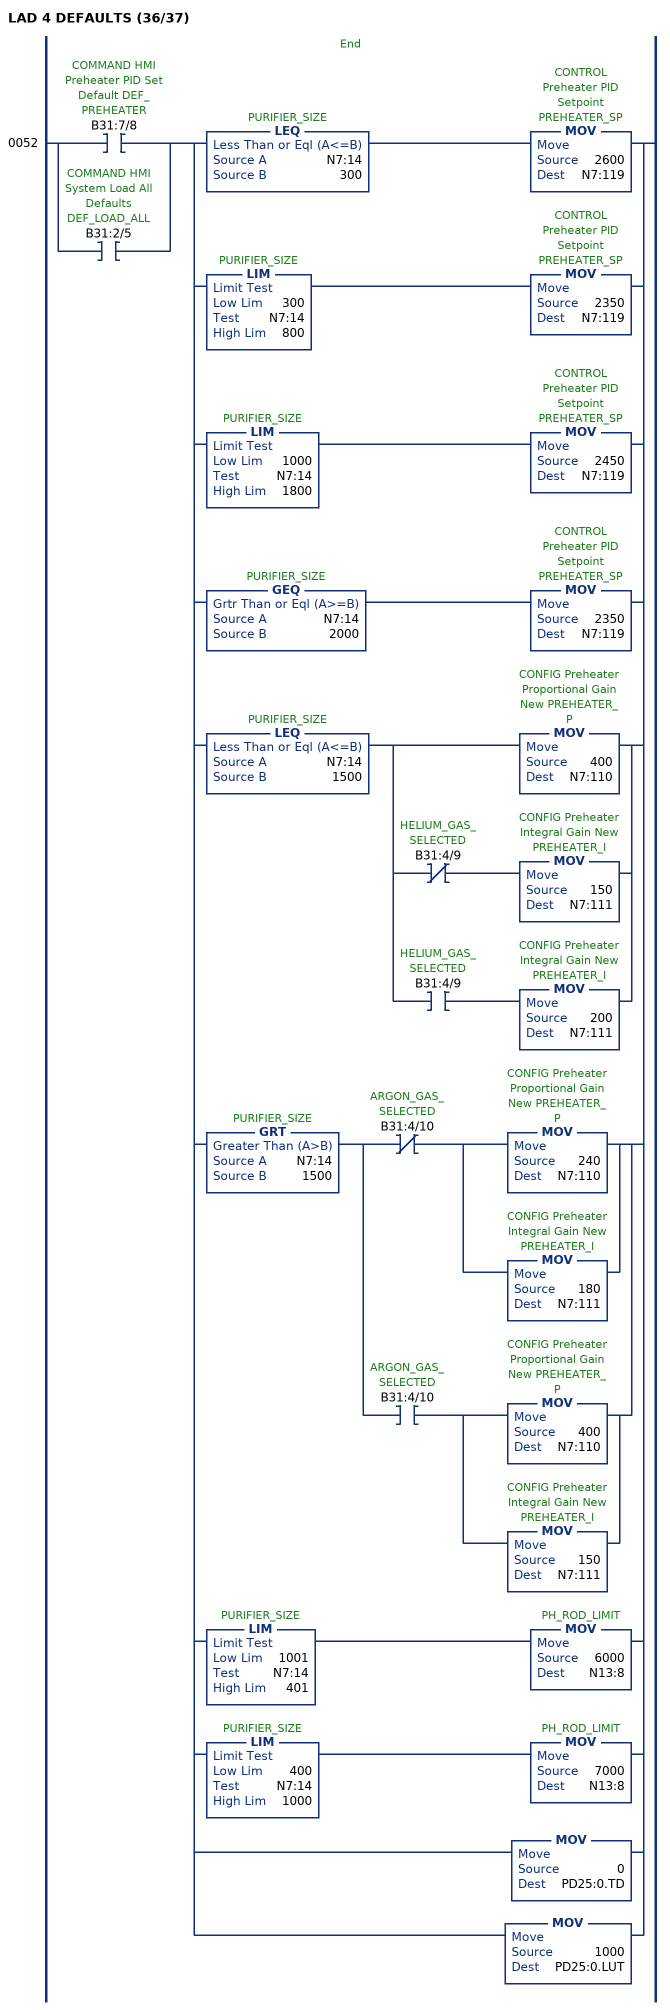
% Rung: 52 %
% End %
SOR BST XIC B31:7/8 NXB XIC B31:2/5 BND BST BST LEQ N7:14 300 MOV 2600 N7:119 NXB LIM 300 N7:14 800 MOV 2350 N7:119 NXB LIM 1000 N7:14 1800 MOV 2450 N7:119 NXB GEQ N7:14 2000 MOV 2350 N7:119 BND NXB BST LEQ N7:14 1500 BST MOV 400 N7:110 NXB BST XIO B31:4/9 MOV 150 N7:111 NXB XIC B31:4/9 MOV 200 N7:111 BND BND NXB GRT N7:14 1500 BST XIO B31:4/10 BST MOV 240 N7:110 NXB MOV 180 N7:111 BND NXB XIC B31:4/10 BST MOV 400 N7:110 NXB MOV 150 N7:111 BND BND BND NXB BST LIM 1001 N7:14 401 MOV 6000 N13:8 NXB LIM 400 N7:14 1000 MOV 7000 N13:8 BND NXB MOV 0 PD25:0.TD NXB MOV 1000 PD25:0.LUT BND EOR
%   B31:7/8  DEF_PREHEATER  "COMMAND HMI Preheater PID Set Default" %
%   B31:2/5  DEF_LOAD_ALL  "COMMAND HMI System Load All Defaults" %
%   N7:14  PURIFIER_SIZE %
%   N7:119  PREHEATER_SP  "CONTROL Preheater PID Setpoint" %
%   N7:110  PREHEATER_P  "CONFIG Preheater Proportional Gain New" %
%   B31:4/9  HELIUM_GAS_SELECTED %
%   N7:111  PREHEATER_I  "CONFIG Preheater Integral Gain New" %
%   B31:4/10  ARGON_GAS_SELECTED %
%   N13:8  PH_ROD_LIMIT %

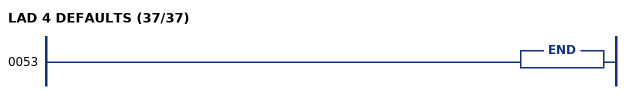
% Rung: 53 %
SOR END EOR

LADDER 5 "SYS_FAULTS"    % Monitors the system fault conditions %
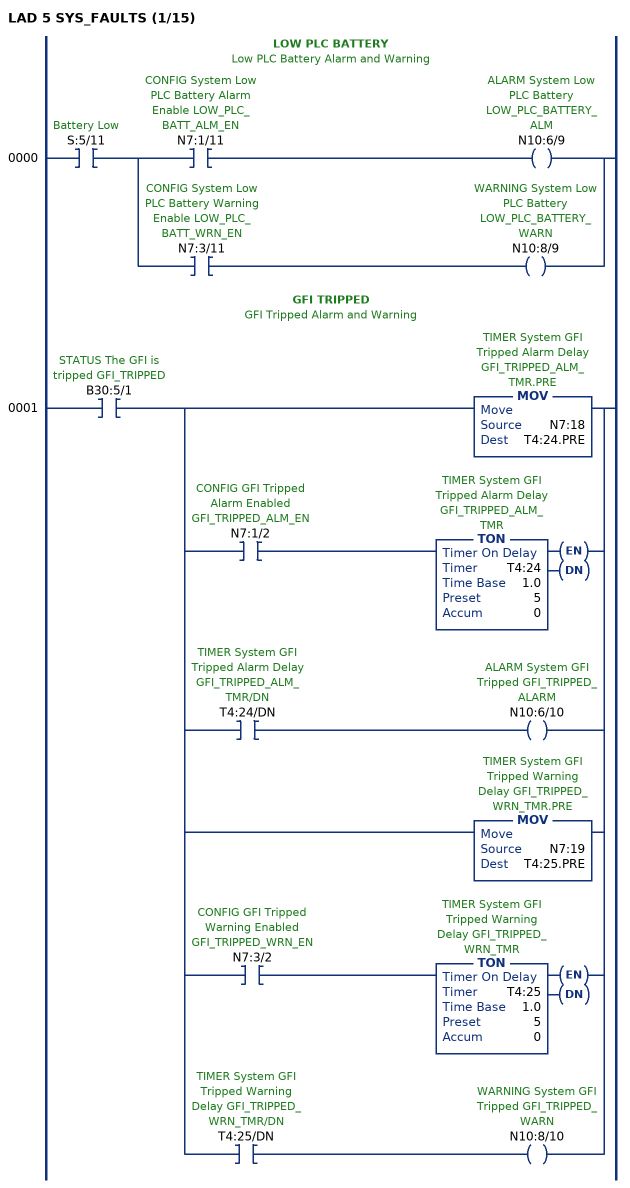
% Rung: 0 %
% TITLE: LOW PLC BATTERY %
% Low PLC Battery Alarm and Warning %
SOR XIC S:5/11 BST XIC N7:1/11 OTE N10:6/9 NXB XIC N7:3/11 OTE N10:8/9 BND EOR
%   S:5/11  "Battery Low" %
%   N7:1/11  LOW_PLC_BATT_ALM_EN  "CONFIG System Low PLC Battery Alarm Enable" %
%   N10:6/9  LOW_PLC_BATTERY_ALM  "ALARM System Low PLC Battery" %
%   N7:3/11  LOW_PLC_BATT_WRN_EN  "CONFIG System Low PLC Battery Warning Enable" %
%   N10:8/9  LOW_PLC_BATTERY_WARN  "WARNING System Low PLC Battery" %
% Rung: 1 %
% TITLE: GFI TRIPPED %
% GFI Tripped Alarm and Warning %
SOR XIC B30:5/1 BST MOV N7:18 T4:24.PRE NXB XIC N7:1/2 TON T4:24 1.0 5 0 NXB XIC T4:24/DN OTE N10:6/10 NXB MOV N7:19 T4:25.PRE NXB XIC N7:3/2 TON T4:25 1.0 5 0 NXB XIC T4:25/DN OTE N10:8/10 BND EOR
%   B30:5/1  GFI_TRIPPED  "STATUS The GFI is tripped" %
%   N7:18  GFI_TRIPPED_ALM_DLY  "CONFIG GFI fault alarm delay" %
%   T4:24  GFI_TRIPPED_ALM_TMR  "TIMER System GFI Tripped Alarm Delay" %
%   N7:1/2  GFI_TRIPPED_ALM_EN  "CONFIG GFI Tripped Alarm Enabled" %
%   N10:6/10  GFI_TRIPPED_ALARM  "ALARM System GFI Tripped" %
%   N7:19  GFI_TRIPPED_WRN_DLY  "CONFIG GFI fault warning delay" %
%   T4:25  GFI_TRIPPED_WRN_TMR  "TIMER System GFI Tripped Warning Delay" %
%   N7:3/2  GFI_TRIPPED_WRN_EN  "CONFIG GFI Tripped Warning Enabled" %
%   N10:8/10  GFI_TRIPPED_WARN  "WARNING System GFI Tripped" %

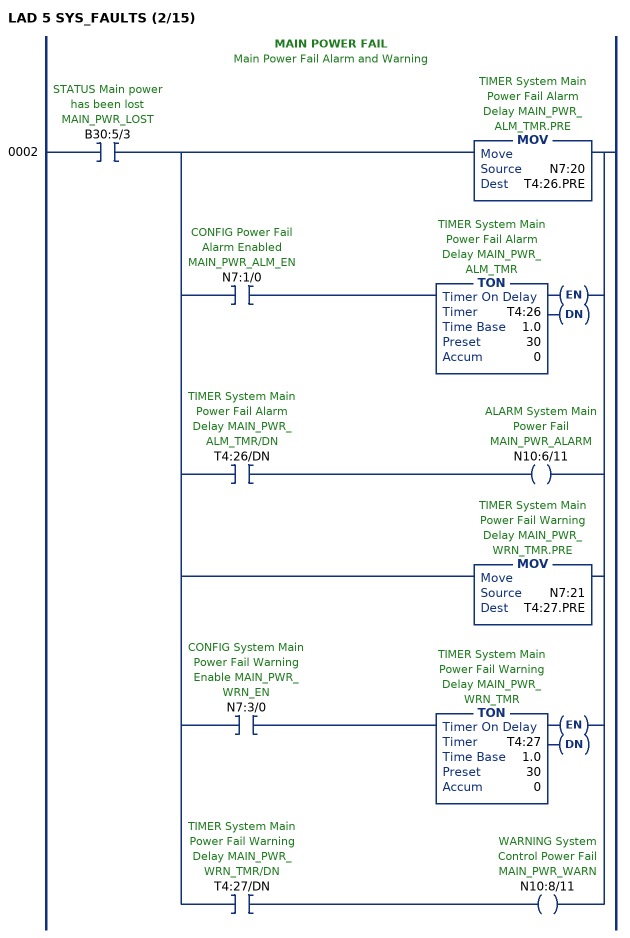
% Rung: 2 %
% TITLE: MAIN POWER FAIL %
% Main Power Fail Alarm and Warning %
SOR XIC B30:5/3 BST MOV N7:20 T4:26.PRE NXB XIC N7:1/0 TON T4:26 1.0 30 0 NXB XIC T4:26/DN OTE N10:6/11 NXB MOV N7:21 T4:27.PRE NXB XIC N7:3/0 TON T4:27 1.0 30 0 NXB XIC T4:27/DN OTE N10:8/11 BND EOR
%   B30:5/3  MAIN_PWR_LOST  "STATUS Main power has been lost" %
%   N7:20  PWR_FAIL_ALM_DELAY  "CONFIG System Power failure Alarm Delay" %
%   T4:26  MAIN_PWR_ALM_TMR  "TIMER System Main Power Fail Alarm Delay" %
%   N7:1/0  MAIN_PWR_ALM_EN  "CONFIG Power Fail Alarm Enabled" %
%   N10:6/11  MAIN_PWR_ALARM  "ALARM System Main Power Fail" %
%   N7:21  PWR_FAIL_WRN_DELAY  "CONFIG System Power Failure Warning Delay" %
%   T4:27  MAIN_PWR_WRN_TMR  "TIMER System Main Power Fail Warning Delay" %
%   N7:3/0  MAIN_PWR_WRN_EN  "CONFIG System Main Power Fail Warning Enable" %
%   N10:8/11  MAIN_PWR_WARN  "WARNING System Control Power Fail" %

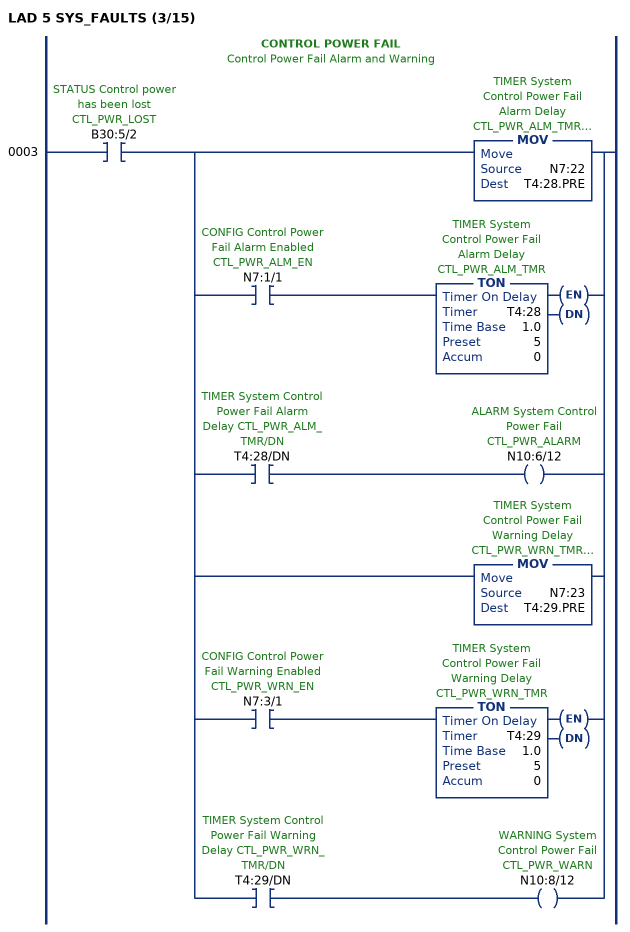
% Rung: 3 %
% TITLE: CONTROL POWER FAIL %
% Control Power Fail Alarm and Warning %
SOR XIC B30:5/2 BST MOV N7:22 T4:28.PRE NXB XIC N7:1/1 TON T4:28 1.0 5 0 NXB XIC T4:28/DN OTE N10:6/12 NXB MOV N7:23 T4:29.PRE NXB XIC N7:3/1 TON T4:29 1.0 5 0 NXB XIC T4:29/DN OTE N10:8/12 BND EOR
%   B30:5/2  CTL_PWR_LOST  "STATUS Control power has been lost" %
%   N7:22  CTL_PWR_FAIL_ALM_DLY  "CONFIG Control power alarm delay setpoint" %
%   T4:28  CTL_PWR_ALM_TMR  "TIMER System Control Power Fail Alarm Delay" %
%   N7:1/1  CTL_PWR_ALM_EN  "CONFIG Control Power Fail Alarm Enabled" %
%   N10:6/12  CTL_PWR_ALARM  "ALARM System Control Power Fail" %
%   N7:23  CTL_PWR_FAIL_WRN_DLY  "CONFIG Control power failure warning delay setpoint" %
%   T4:29  CTL_PWR_WRN_TMR  "TIMER System Control Power Fail Warning Delay" %
%   N7:3/1  CTL_PWR_WRN_EN  "CONFIG Control Power Fail Warning Enabled" %
%   N10:8/12  CTL_PWR_WARN  "WARNING System Control Power Fail" %

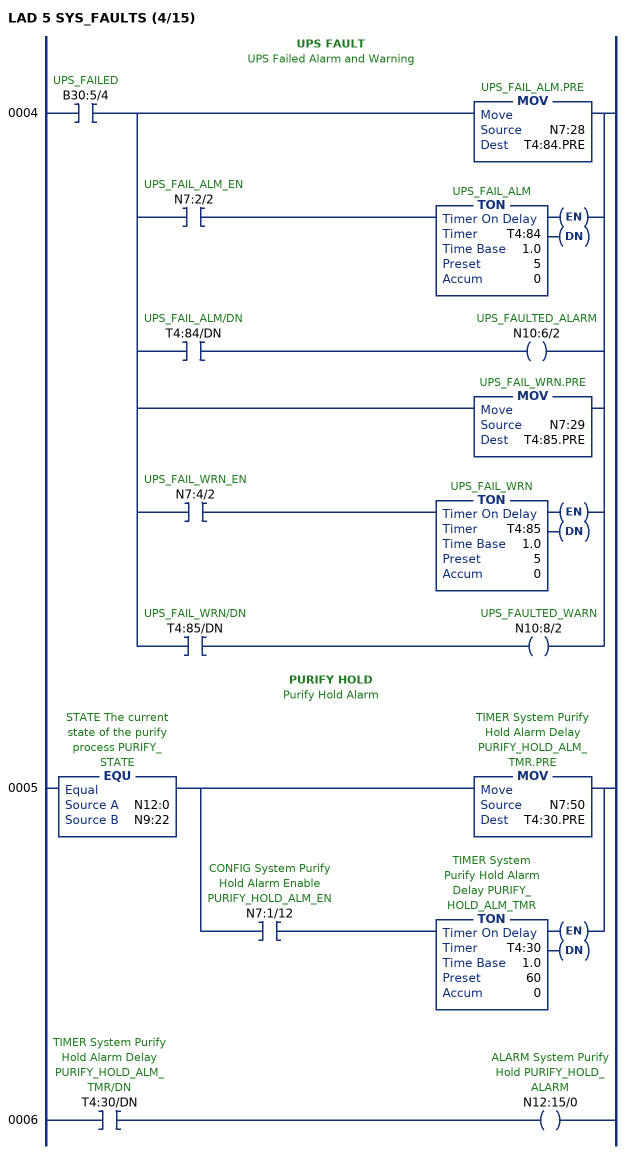
% Rung: 4 %
% TITLE: UPS FAULT %
% UPS Failed Alarm and Warning %
SOR XIC B30:5/4 BST MOV N7:28 T4:84.PRE NXB XIC N7:2/2 TON T4:84 1.0 5 0 NXB XIC T4:84/DN OTE N10:6/2 NXB MOV N7:29 T4:85.PRE NXB XIC N7:4/2 TON T4:85 1.0 5 0 NXB XIC T4:85/DN OTE N10:8/2 BND EOR
%   B30:5/4  UPS_FAILED %
%   N7:28  UPS_FAIL_ALM_DLY %
%   T4:84  UPS_FAIL_ALM %
%   N7:2/2  UPS_FAIL_ALM_EN %
%   N10:6/2  UPS_FAULTED_ALARM %
%   N7:29  UPS_FAIL_WRN_DLY %
%   T4:85  UPS_FAIL_WRN %
%   N7:4/2  UPS_FAIL_WRN_EN %
%   N10:8/2  UPS_FAULTED_WARN %
% Rung: 5 %
% TITLE: PURIFY HOLD %
% Purify Hold Alarm %
SOR EQU N12:0 N9:22 BST MOV N7:50 T4:30.PRE NXB XIC N7:1/12 TON T4:30 1.0 60 0 BND EOR
%   N12:0  PURIFY_STATE  "STATE The current state of the purify process" %
%   N9:22  PURIFY_HOLD  "STATE Purify Hold" %
%   N7:50  PURIFY_HOLD_ALM_DLY  "CONFIG System Purify Hold Alarm Delay" %
%   T4:30  PURIFY_HOLD_ALM_TMR  "TIMER System Purify Hold Alarm Delay" %
%   N7:1/12  PURIFY_HOLD_ALM_EN  "CONFIG System Purify Hold Alarm Enable" %
% Rung: 6 %
SOR XIC T4:30/DN OTE N12:15/0 EOR
%   T4:30  PURIFY_HOLD_ALM_TMR  "TIMER System Purify Hold Alarm Delay" %
%   N12:15/0  PURIFY_HOLD_ALARM  "ALARM System Purify Hold" %

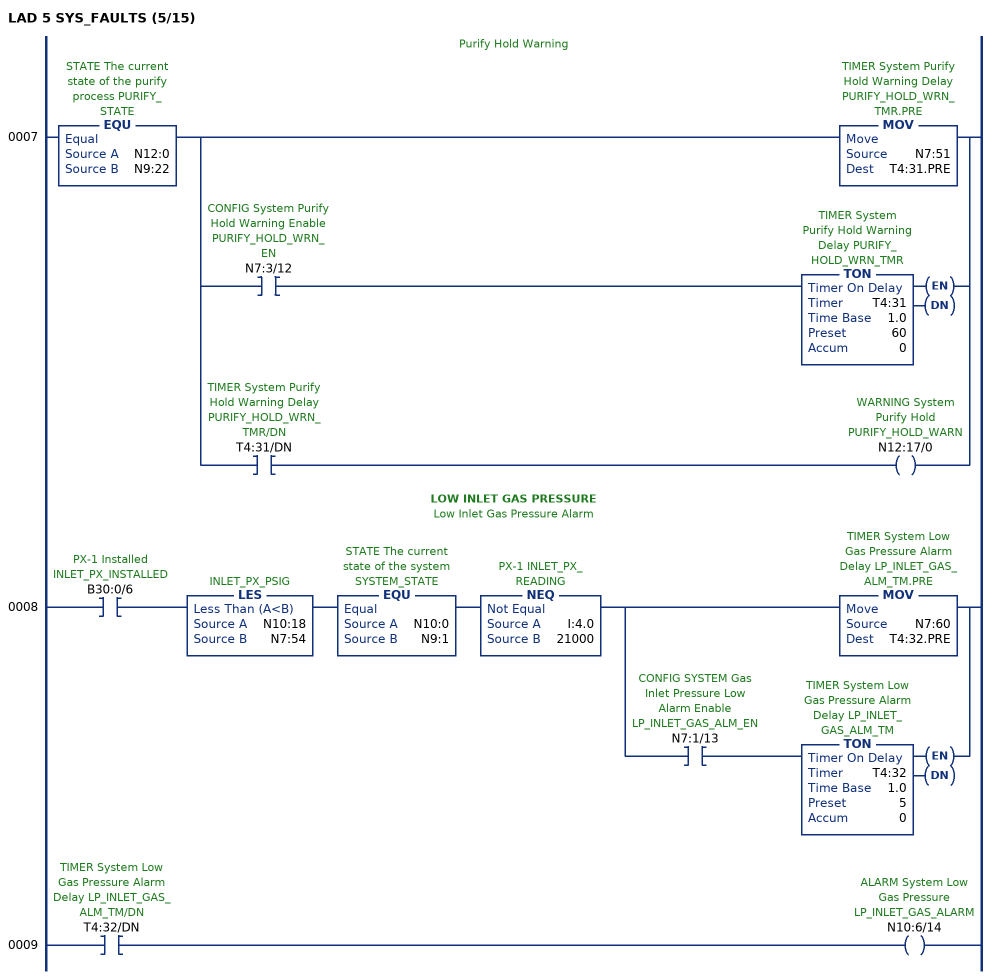
% Rung: 7 %
% Purify Hold Warning %
SOR EQU N12:0 N9:22 BST MOV N7:51 T4:31.PRE NXB XIC N7:3/12 TON T4:31 1.0 60 0 NXB XIC T4:31/DN OTE N12:17/0 BND EOR
%   N12:0  PURIFY_STATE  "STATE The current state of the purify process" %
%   N9:22  PURIFY_HOLD  "STATE Purify Hold" %
%   N7:51  PURIFY_HOLD_WRN_DLY  "CONFIG System Purify Hold Warning Delay" %
%   T4:31  PURIFY_HOLD_WRN_TMR  "TIMER System Purify Hold Warning Delay" %
%   N7:3/12  PURIFY_HOLD_WRN_EN  "CONFIG System Purify Hold Warning Enable" %
%   N12:17/0  PURIFY_HOLD_WARN  "WARNING System Purify Hold" %
% Rung: 8 %
% TITLE: LOW INLET GAS PRESSURE %
% Low Inlet Gas Pressure Alarm %
SOR XIC B30:0/6 LES N10:18 N7:54 EQU N10:0 N9:1 NEQ I:4.0 21000 BST MOV N7:60 T4:32.PRE NXB XIC N7:1/13 TON T4:32 1.0 5 0 BND EOR
%   B30:0/6  INLET_PX_INSTALLED  "PX-1 Installed" %
%   N10:18  INLET_PX_PSIG %
%   N7:54  LP_INLET_GAS_ALM_SP  "CONFIG SYSTEM Gas Inlet Pressure Low Alarm Setpoint" %
%   N10:0  SYSTEM_STATE  "STATE The current state of the system" %
%   N9:1  SYSTEM_PROCESS  "STATE System Process" %
%   I:4.0  INLET_PX_READING  "PX-1" %
%   N7:60  LP_INLET_GAS_ALM_DLY  "CONFIG SYSTEM Gas Inlet Pressure Low Alarm Delay" %
%   T4:32  LP_INLET_GAS_ALM_TM  "TIMER System Low Gas Pressure Alarm Delay" %
%   N7:1/13  LP_INLET_GAS_ALM_EN  "CONFIG SYSTEM Gas Inlet Pressure Low Alarm Enable" %
% Rung: 9 %
SOR XIC T4:32/DN OTE N10:6/14 EOR
%   T4:32  LP_INLET_GAS_ALM_TM  "TIMER System Low Gas Pressure Alarm Delay" %
%   N10:6/14  LP_INLET_GAS_ALARM  "ALARM System Low Gas Pressure" %

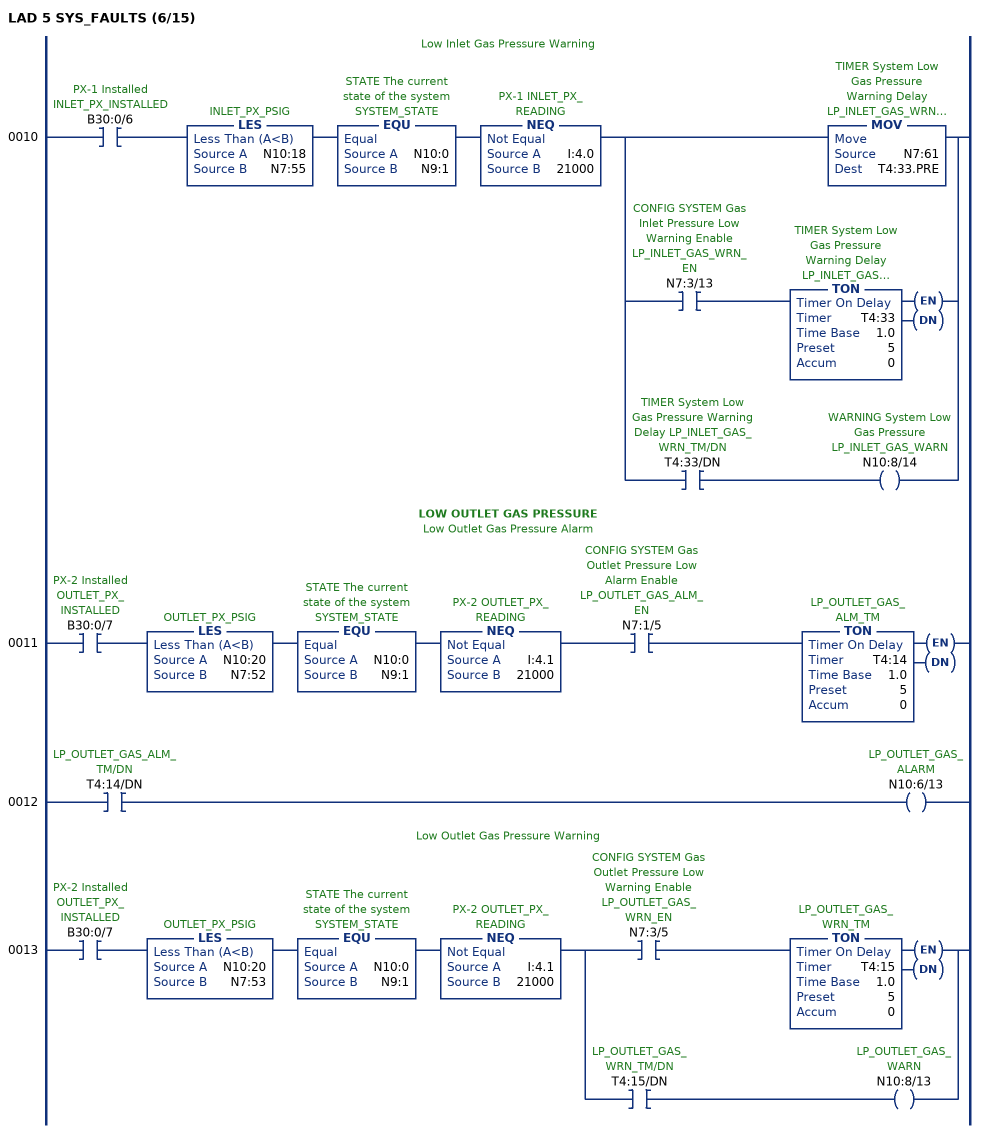
% Rung: 10 %
% Low Inlet Gas Pressure Warning %
SOR XIC B30:0/6 LES N10:18 N7:55 EQU N10:0 N9:1 NEQ I:4.0 21000 BST MOV N7:61 T4:33.PRE NXB XIC N7:3/13 TON T4:33 1.0 5 0 NXB XIC T4:33/DN OTE N10:8/14 BND EOR
%   B30:0/6  INLET_PX_INSTALLED  "PX-1 Installed" %
%   N10:18  INLET_PX_PSIG %
%   N7:55  LP_INLET_GAS_WRN_SP  "CONFIG SYSTEM Gas Inlet Pressure Low Warning Setpoint" %
%   N10:0  SYSTEM_STATE  "STATE The current state of the system" %
%   N9:1  SYSTEM_PROCESS  "STATE System Process" %
%   I:4.0  INLET_PX_READING  "PX-1" %
%   N7:61  LP_INLET_GAS_WRN_DLY  "CONFIG SYSTEM Gas Inlet Pressure Low Warning Delay" %
%   T4:33  LP_INLET_GAS_WRN_TM  "TIMER System Low Gas Pressure Warning Delay" %
%   N7:3/13  LP_INLET_GAS_WRN_EN  "CONFIG SYSTEM Gas Inlet Pressure Low Warning Enable" %
%   N10:8/14  LP_INLET_GAS_WARN  "WARNING System Low Gas Pressure" %
% Rung: 11 %
% TITLE: LOW OUTLET GAS PRESSURE %
% Low Outlet Gas Pressure Alarm %
SOR XIC B30:0/7 LES N10:20 N7:52 EQU N10:0 N9:1 NEQ I:4.1 21000 XIC N7:1/5 TON T4:14 1.0 5 0 EOR
%   B30:0/7  OUTLET_PX_INSTALLED  "PX-2 Installed" %
%   N10:20  OUTLET_PX_PSIG %
%   N7:52  LP_OUTLET_GAS_ALM_SP  "CONFIG SYSTEM Gas Outlet Pressure Low Alarm Setpoint" %
%   N10:0  SYSTEM_STATE  "STATE The current state of the system" %
%   N9:1  SYSTEM_PROCESS  "STATE System Process" %
%   I:4.1  OUTLET_PX_READING  "PX-2" %
%   N7:1/5  LP_OUTLET_GAS_ALM_EN  "CONFIG SYSTEM Gas Outlet Pressure Low Alarm Enable" %
%   T4:14  LP_OUTLET_GAS_ALM_TM %
% Rung: 12 %
SOR XIC T4:14/DN OTE N10:6/13 EOR
%   T4:14  LP_OUTLET_GAS_ALM_TM %
%   N10:6/13  LP_OUTLET_GAS_ALARM %
% Rung: 13 %
% Low Outlet Gas Pressure Warning %
SOR XIC B30:0/7 LES N10:20 N7:53 EQU N10:0 N9:1 NEQ I:4.1 21000 BST XIC N7:3/5 TON T4:15 1.0 5 0 NXB XIC T4:15/DN OTE N10:8/13 BND EOR
%   B30:0/7  OUTLET_PX_INSTALLED  "PX-2 Installed" %
%   N10:20  OUTLET_PX_PSIG %
%   N7:53  LP_OUTLET_GAS_WRN_SP  "CONFIG SYSTEM Gas Outlet Pressure Low Warning Setpoint" %
%   N10:0  SYSTEM_STATE  "STATE The current state of the system" %
%   N9:1  SYSTEM_PROCESS  "STATE System Process" %
%   I:4.1  OUTLET_PX_READING  "PX-2" %
%   N7:3/5  LP_OUTLET_GAS_WRN_EN  "CONFIG SYSTEM Gas Outlet Pressure Low Warning Enable" %
%   T4:15  LP_OUTLET_GAS_WRN_TM %
%   N10:8/13  LP_OUTLET_GAS_WARN %

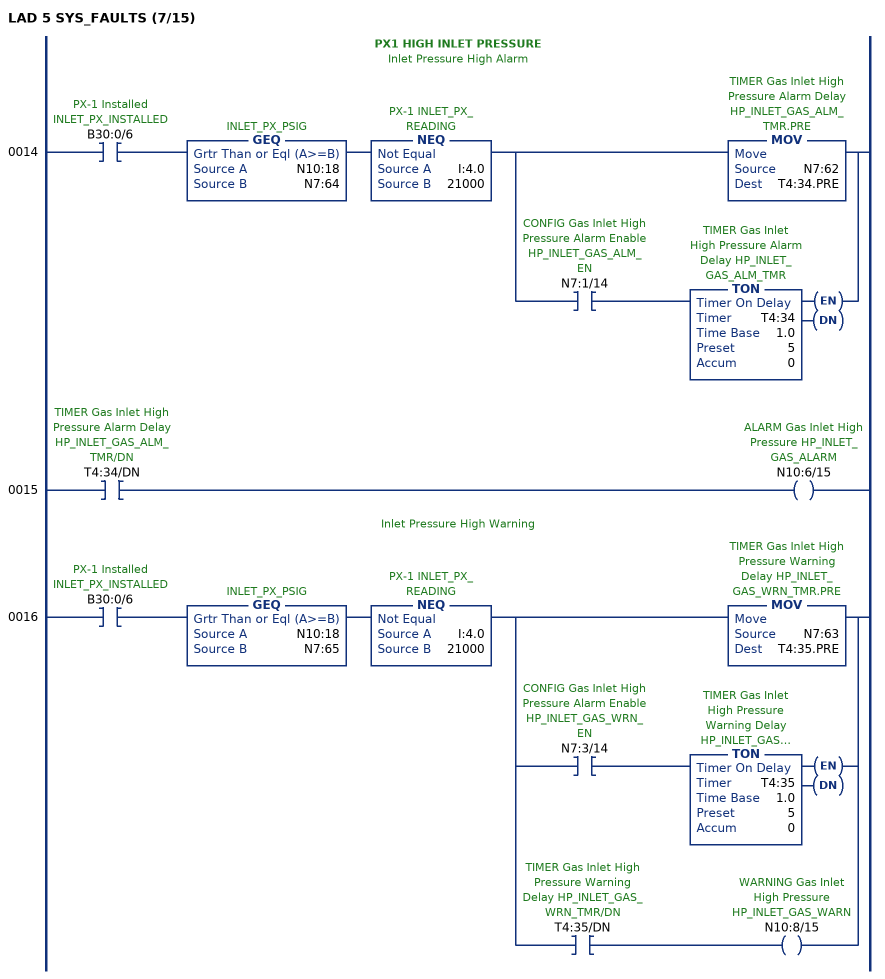
% Rung: 14 %
% TITLE: PX1 HIGH INLET PRESSURE %
% Inlet Pressure High Alarm %
SOR XIC B30:0/6 GEQ N10:18 N7:64 NEQ I:4.0 21000 BST MOV N7:62 T4:34.PRE NXB XIC N7:1/14 TON T4:34 1.0 5 0 BND EOR
%   B30:0/6  INLET_PX_INSTALLED  "PX-1 Installed" %
%   N10:18  INLET_PX_PSIG %
%   N7:64  HP_INLET_GAS_ALM_SP  "CONFIG Gas Inlet High Pressure Alarm Setpoint" %
%   I:4.0  INLET_PX_READING  "PX-1" %
%   N7:62  HP_INLET_GAS_ALM_DLY  "CONFIG Gas Inlet High Pressure Alarm Delay" %
%   T4:34  HP_INLET_GAS_ALM_TMR  "TIMER Gas Inlet High Pressure Alarm Delay" %
%   N7:1/14  HP_INLET_GAS_ALM_EN  "CONFIG Gas Inlet High Pressure Alarm Enable" %
% Rung: 15 %
SOR XIC T4:34/DN OTE N10:6/15 EOR
%   T4:34  HP_INLET_GAS_ALM_TMR  "TIMER Gas Inlet High Pressure Alarm Delay" %
%   N10:6/15  HP_INLET_GAS_ALARM  "ALARM Gas Inlet High Pressure" %
% Rung: 16 %
% Inlet Pressure High Warning %
SOR XIC B30:0/6 GEQ N10:18 N7:65 NEQ I:4.0 21000 BST MOV N7:63 T4:35.PRE NXB XIC N7:3/14 TON T4:35 1.0 5 0 NXB XIC T4:35/DN OTE N10:8/15 BND EOR
%   B30:0/6  INLET_PX_INSTALLED  "PX-1 Installed" %
%   N10:18  INLET_PX_PSIG %
%   N7:65  HP_INLET_GAS_WRN_SP  "CONFIG Gas Inlet High Pressure Warning Setpoint" %
%   I:4.0  INLET_PX_READING  "PX-1" %
%   N7:63  HP_INLET_GAS_WRN_DLY  "CONFIG Gas Inlet High Pressure Warning Delay" %
%   T4:35  HP_INLET_GAS_WRN_TMR  "TIMER Gas Inlet High Pressure Warning Delay" %
%   N7:3/14  HP_INLET_GAS_WRN_EN  "CONFIG Gas Inlet High Pressure Alarm Enable" %
%   N10:8/15  HP_INLET_GAS_WARN  "WARNING Gas Inlet High Pressure" %

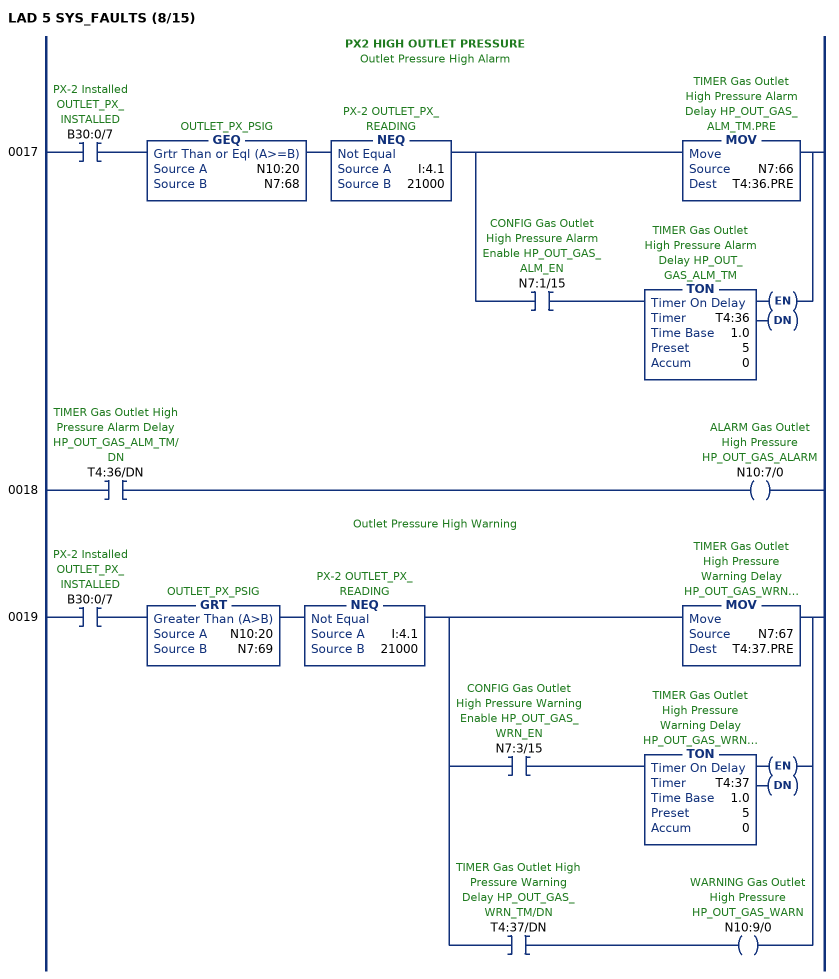
% Rung: 17 %
% TITLE: PX2 HIGH OUTLET PRESSURE %
% Outlet Pressure High Alarm %
SOR XIC B30:0/7 GEQ N10:20 N7:68 NEQ I:4.1 21000 BST MOV N7:66 T4:36.PRE NXB XIC N7:1/15 TON T4:36 1.0 5 0 BND EOR
%   B30:0/7  OUTLET_PX_INSTALLED  "PX-2 Installed" %
%   N10:20  OUTLET_PX_PSIG %
%   N7:68  HP_OUT_GAS_ALM_SP  "CONFIG Gas Outlet High Pressure Alarm Setpoint" %
%   I:4.1  OUTLET_PX_READING  "PX-2" %
%   N7:66  HP_OUT_GAS_ALM_DLY  "CONFIG Gas Outlet High Pressure Alarm Deley" %
%   T4:36  HP_OUT_GAS_ALM_TM  "TIMER Gas Outlet High Pressure Alarm Delay" %
%   N7:1/15  HP_OUT_GAS_ALM_EN  "CONFIG Gas Outlet High Pressure Alarm Enable" %
% Rung: 18 %
SOR XIC T4:36/DN OTE N10:7/0 EOR
%   T4:36  HP_OUT_GAS_ALM_TM  "TIMER Gas Outlet High Pressure Alarm Delay" %
%   N10:7/0  HP_OUT_GAS_ALARM  "ALARM Gas Outlet High Pressure" %
% Rung: 19 %
% Outlet Pressure High Warning %
SOR XIC B30:0/7 GRT N10:20 N7:69 NEQ I:4.1 21000 BST MOV N7:67 T4:37.PRE NXB XIC N7:3/15 TON T4:37 1.0 5 0 NXB XIC T4:37/DN OTE N10:9/0 BND EOR
%   B30:0/7  OUTLET_PX_INSTALLED  "PX-2 Installed" %
%   N10:20  OUTLET_PX_PSIG %
%   N7:69  HP_OUT_GAS_WRN_SP  "CONFIG Gas Outlet High Pressure Warning Setpoint" %
%   I:4.1  OUTLET_PX_READING  "PX-2" %
%   N7:67  HP_OUT_GAS_WRN_DLY  "CONFIG Gas Outlet High Pressure Warning Delay" %
%   T4:37  HP_OUT_GAS_WRN_TM  "TIMER Gas Outlet High Pressure Warning Delay" %
%   N7:3/15  HP_OUT_GAS_WRN_EN  "CONFIG Gas Outlet High Pressure Warning Enable" %
%   N10:9/0  HP_OUT_GAS_WARN  "WARNING Gas Outlet High Pressure" %

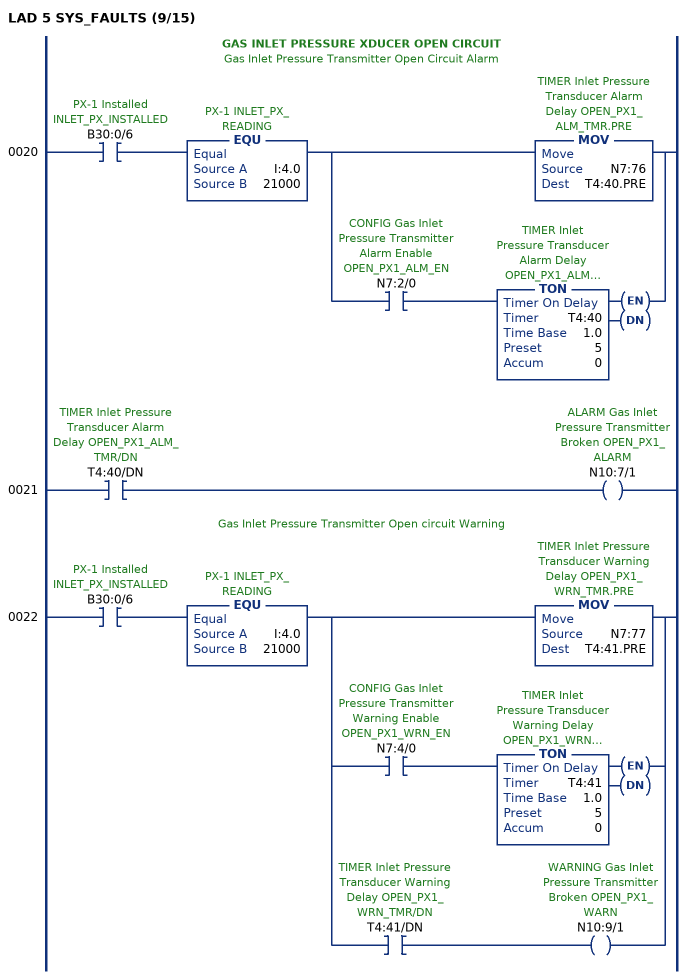
% Rung: 20 %
% TITLE: GAS INLET PRESSURE XDUCER OPEN CIRCUIT %
% Gas Inlet Pressure Transmitter Open Circuit Alarm %
SOR XIC B30:0/6 EQU I:4.0 21000 BST MOV N7:76 T4:40.PRE NXB XIC N7:2/0 TON T4:40 1.0 5 0 BND EOR
%   B30:0/6  INLET_PX_INSTALLED  "PX-1 Installed" %
%   I:4.0  INLET_PX_READING  "PX-1" %
%   N7:76  OPEN_PX1_ALM_DLY  "CONFIG Gas Inlet Pressure Transducer Alarm Delay" %
%   T4:40  OPEN_PX1_ALM_TMR  "TIMER Inlet Pressure Transducer Alarm Delay" %
%   N7:2/0  OPEN_PX1_ALM_EN  "CONFIG Gas Inlet Pressure Transmitter Alarm Enable" %
% Rung: 21 %
SOR XIC T4:40/DN OTE N10:7/1 EOR
%   T4:40  OPEN_PX1_ALM_TMR  "TIMER Inlet Pressure Transducer Alarm Delay" %
%   N10:7/1  OPEN_PX1_ALARM  "ALARM Gas Inlet Pressure Transmitter Broken" %
% Rung: 22 %
% Gas Inlet Pressure Transmitter Open circuit Warning %
SOR XIC B30:0/6 EQU I:4.0 21000 BST MOV N7:77 T4:41.PRE NXB XIC N7:4/0 TON T4:41 1.0 5 0 NXB XIC T4:41/DN OTE N10:9/1 BND EOR
%   B30:0/6  INLET_PX_INSTALLED  "PX-1 Installed" %
%   I:4.0  INLET_PX_READING  "PX-1" %
%   N7:77  OPEN_PX1_WRN_DLY  "CONFIG Gas Inlet Pressure Transducer Warning Delay" %
%   T4:41  OPEN_PX1_WRN_TMR  "TIMER Inlet Pressure Transducer Warning Delay" %
%   N7:4/0  OPEN_PX1_WRN_EN  "CONFIG Gas Inlet Pressure Transmitter Warning Enable" %
%   N10:9/1  OPEN_PX1_WARN  "WARNING Gas Inlet Pressure Transmitter Broken" %

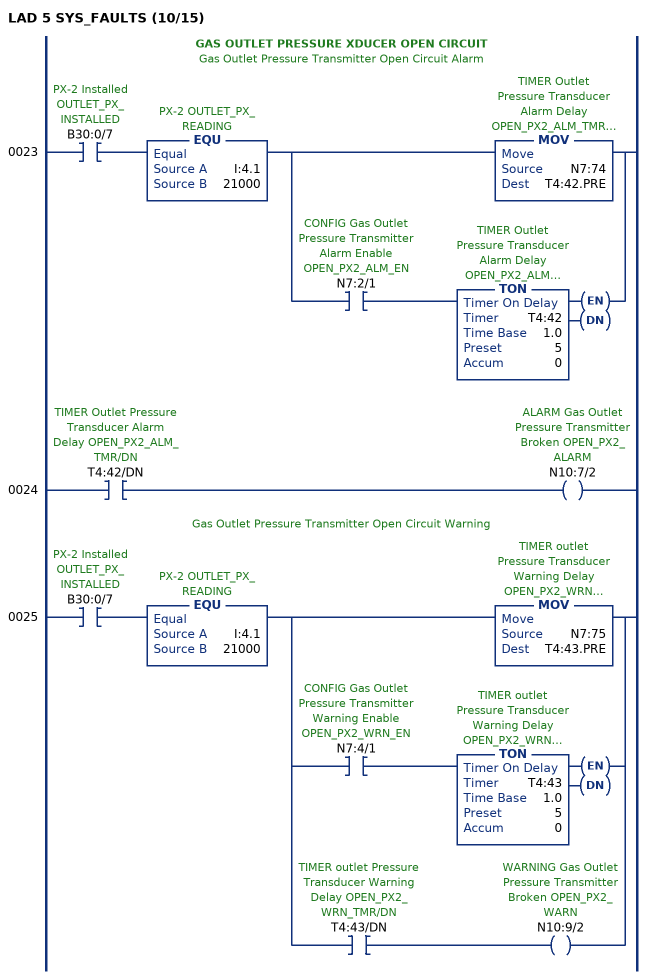
% Rung: 23 %
% TITLE: GAS OUTLET PRESSURE XDUCER OPEN CIRCUIT %
% Gas Outlet Pressure Transmitter Open Circuit Alarm %
SOR XIC B30:0/7 EQU I:4.1 21000 BST MOV N7:74 T4:42.PRE NXB XIC N7:2/1 TON T4:42 1.0 5 0 BND EOR
%   B30:0/7  OUTLET_PX_INSTALLED  "PX-2 Installed" %
%   I:4.1  OUTLET_PX_READING  "PX-2" %
%   N7:74  OPEN_PX2_ALM_DLY  "CONFIG Gas Outlet Pressure Transducer Alarm Delay" %
%   T4:42  OPEN_PX2_ALM_TMR  "TIMER Outlet Pressure Transducer Alarm Delay" %
%   N7:2/1  OPEN_PX2_ALM_EN  "CONFIG Gas Outlet Pressure Transmitter Alarm Enable" %
% Rung: 24 %
SOR XIC T4:42/DN OTE N10:7/2 EOR
%   T4:42  OPEN_PX2_ALM_TMR  "TIMER Outlet Pressure Transducer Alarm Delay" %
%   N10:7/2  OPEN_PX2_ALARM  "ALARM Gas Outlet Pressure Transmitter Broken" %
% Rung: 25 %
% Gas Outlet Pressure Transmitter Open Circuit Warning %
SOR XIC B30:0/7 EQU I:4.1 21000 BST MOV N7:75 T4:43.PRE NXB XIC N7:4/1 TON T4:43 1.0 5 0 NXB XIC T4:43/DN OTE N10:9/2 BND EOR
%   B30:0/7  OUTLET_PX_INSTALLED  "PX-2 Installed" %
%   I:4.1  OUTLET_PX_READING  "PX-2" %
%   N7:75  OPEN_PX2_WRN_DLY  "CONFIG Gas Outlet Pressure Transducer Warning Delay" %
%   T4:43  OPEN_PX2_WRN_TMR  "TIMER outlet Pressure Transducer Warning Delay" %
%   N7:4/1  OPEN_PX2_WRN_EN  "CONFIG Gas Outlet Pressure Transmitter Warning Enable" %
%   N10:9/2  OPEN_PX2_WARN  "WARNING Gas Outlet Pressure Transmitter Broken" %

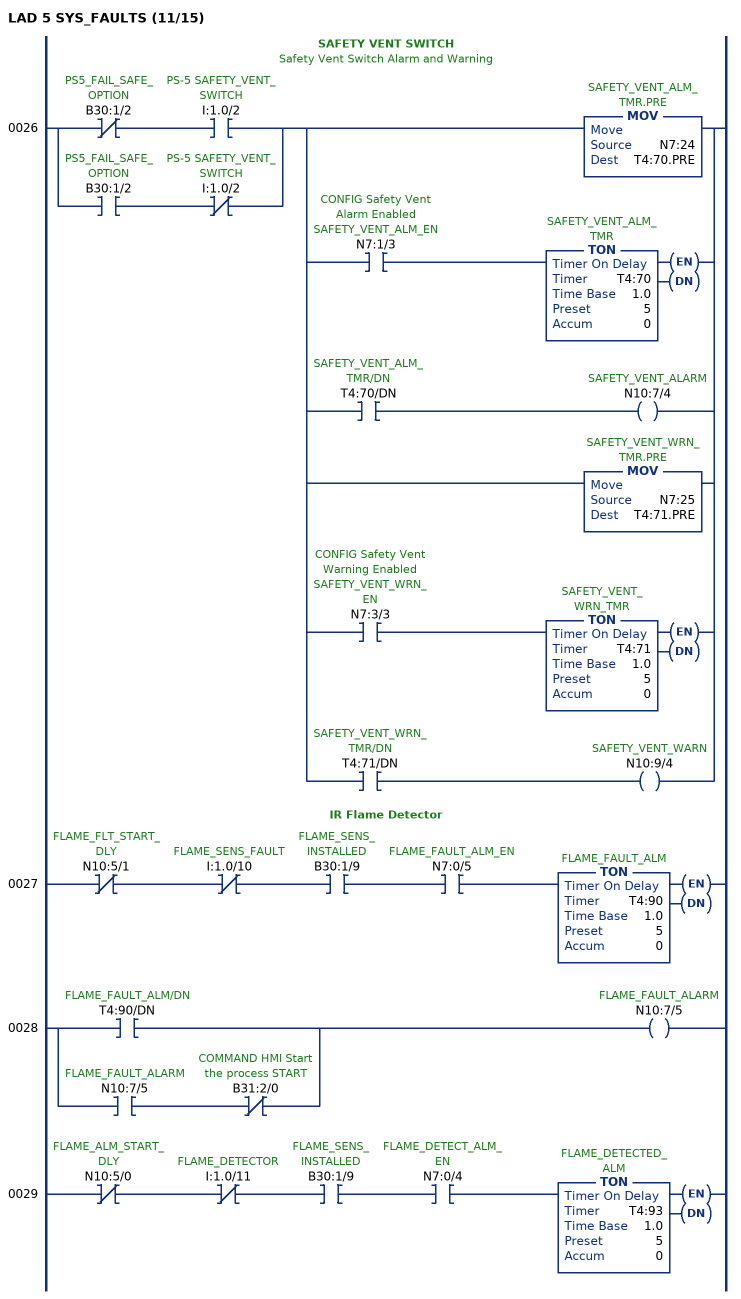
% Rung: 26 %
% TITLE: SAFETY VENT SWITCH %
% Safety Vent Switch Alarm and Warning %
SOR BST XIO B30:1/2 XIC I:1.0/2 NXB XIC B30:1/2 XIO I:1.0/2 BND BST MOV N7:24 T4:70.PRE NXB XIC N7:1/3 TON T4:70 1.0 5 0 NXB XIC T4:70/DN OTE N10:7/4 NXB MOV N7:25 T4:71.PRE NXB XIC N7:3/3 TON T4:71 1.0 5 0 NXB XIC T4:71/DN OTE N10:9/4 BND EOR
%   B30:1/2  PS5_FAIL_SAFE_OPTION %
%   I:1.0/2  SAFETY_VENT_SWITCH  "PS-5" %
%   N7:24  SAFETY_VENT_ALM_DLY  "CONFIG Safety Vent Alarm Delay" %
%   T4:70  SAFETY_VENT_ALM_TMR %
%   N7:1/3  SAFETY_VENT_ALM_EN  "CONFIG Safety Vent Alarm Enabled" %
%   N10:7/4  SAFETY_VENT_ALARM %
%   N7:25  SAFETY_VENT_WRN_DLY  "CONFIG Safety Vent Warning Delay" %
%   T4:71  SAFETY_VENT_WRN_TMR %
%   N7:3/3  SAFETY_VENT_WRN_EN  "CONFIG Safety Vent Warning Enabled" %
%   N10:9/4  SAFETY_VENT_WARN %
% Rung: 27 %
% TITLE: IR Flame Detector %
SOR XIO N10:5/1 XIO I:1.0/10 XIC B30:1/9 XIC N7:0/5 TON T4:90 1.0 5 0 EOR
%   N10:5/1  FLAME_FLT_START_DLY %
%   I:1.0/10  FLAME_SENS_FAULT %
%   B30:1/9  FLAME_SENS_INSTALLED %
%   N7:0/5  FLAME_FAULT_ALM_EN %
%   T4:90  FLAME_FAULT_ALM %
% Rung: 28 %
SOR BST XIC T4:90/DN NXB XIC N10:7/5 XIO B31:2/0 BND OTE N10:7/5 EOR
%   T4:90  FLAME_FAULT_ALM %
%   N10:7/5  FLAME_FAULT_ALARM %
%   B31:2/0  START  "COMMAND HMI Start the process" %
% Rung: 29 %
SOR XIO N10:5/0 XIO I:1.0/11 XIC B30:1/9 XIC N7:0/4 TON T4:93 1.0 5 0 EOR
%   N10:5/0  FLAME_ALM_START_DLY %
%   I:1.0/11  FLAME_DETECTOR %
%   B30:1/9  FLAME_SENS_INSTALLED %
%   N7:0/4  FLAME_DETECT_ALM_EN %
%   T4:93  FLAME_DETECTED_ALM %

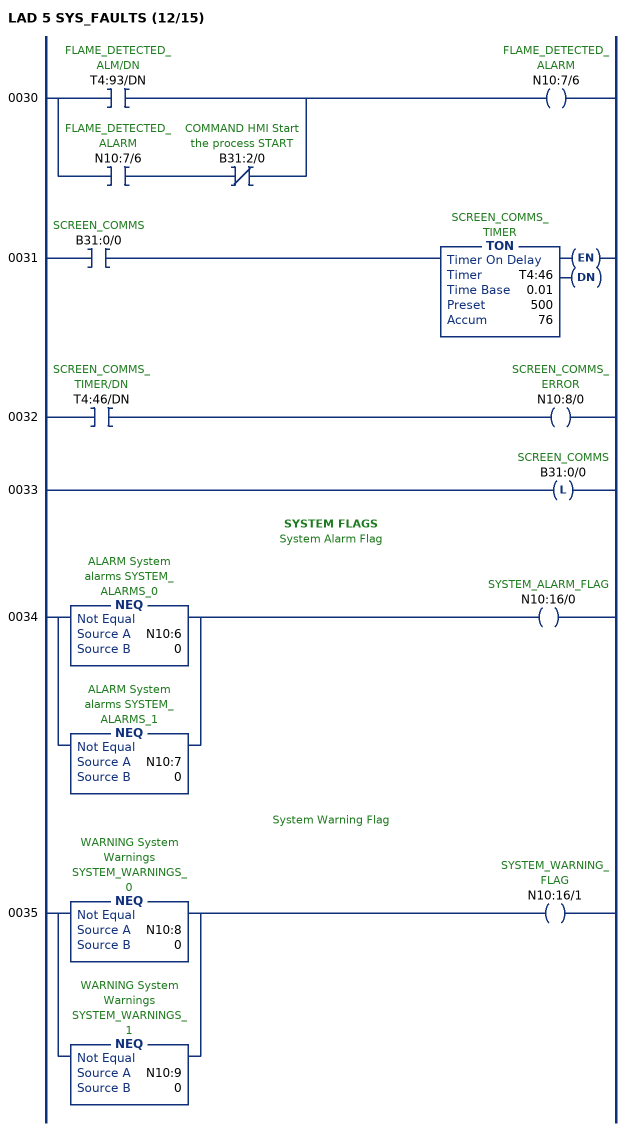
% Rung: 30 %
SOR BST XIC T4:93/DN NXB XIC N10:7/6 XIO B31:2/0 BND OTE N10:7/6 EOR
%   T4:93  FLAME_DETECTED_ALM %
%   N10:7/6  FLAME_DETECTED_ALARM %
%   B31:2/0  START  "COMMAND HMI Start the process" %
% Rung: 31 %
SOR XIC B31:0/0 TON T4:46 0.01 500 76 EOR
%   B31:0/0  SCREEN_COMMS %
%   T4:46  SCREEN_COMMS_TIMER %
% Rung: 32 %
SOR XIC T4:46/DN OTE N10:8/0 EOR
%   T4:46  SCREEN_COMMS_TIMER %
%   N10:8/0  SCREEN_COMMS_ERROR %
% Rung: 33 %
SOR OTL B31:0/0 EOR
%   B31:0/0  SCREEN_COMMS %
% Rung: 34 %
% TITLE: SYSTEM FLAGS %
% System Alarm Flag %
SOR BST NEQ N10:6 0 NXB NEQ N10:7 0 BND OTE N10:16/0 EOR
%   N10:6  SYSTEM_ALARMS_0  "ALARM System alarms" %
%   N10:7  SYSTEM_ALARMS_1  "ALARM System alarms" %
%   N10:16/0  SYSTEM_ALARM_FLAG %
% Rung: 35 %
% System Warning Flag %
SOR BST NEQ N10:8 0 NXB NEQ N10:9 0 BND OTE N10:16/1 EOR
%   N10:8  SYSTEM_WARNINGS_0  "WARNING System Warnings" %
%   N10:9  SYSTEM_WARNINGS_1  "WARNING System Warnings" %
%   N10:16/1  SYSTEM_WARNING_FLAG %

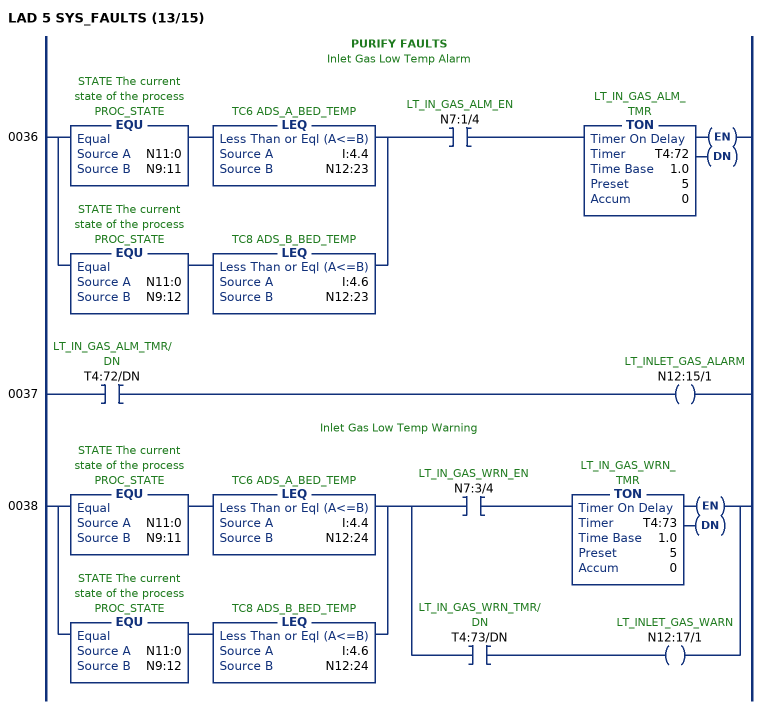
% Rung: 36 %
% TITLE: PURIFY FAULTS %
% Inlet Gas Low Temp Alarm %
SOR BST EQU N11:0 N9:11 LEQ I:4.4 N12:23 NXB EQU N11:0 N9:12 LEQ I:4.6 N12:23 BND XIC N7:1/4 TON T4:72 1.0 5 0 EOR
%   N11:0  PROC_STATE  "STATE The current state of the process" %
%   N9:11  PROC_PURIFY_A  "STATE Process Purify A" %
%   I:4.4  ADS_A_BED_TEMP  "TC6" %
%   N12:23  LT_INLET_GAS_ALM_SP %
%   N9:12  PROC_PURIFY_B  "STATE Process Purify B" %
%   I:4.6  ADS_B_BED_TEMP  "TC8" %
%   N7:1/4  LT_IN_GAS_ALM_EN %
%   T4:72  LT_IN_GAS_ALM_TMR %
% Rung: 37 %
SOR XIC T4:72/DN OTE N12:15/1 EOR
%   T4:72  LT_IN_GAS_ALM_TMR %
%   N12:15/1  LT_INLET_GAS_ALARM %
% Rung: 38 %
% Inlet Gas Low Temp Warning %
SOR BST EQU N11:0 N9:11 LEQ I:4.4 N12:24 NXB EQU N11:0 N9:12 LEQ I:4.6 N12:24 BND BST XIC N7:3/4 TON T4:73 1.0 5 0 NXB XIC T4:73/DN OTE N12:17/1 BND EOR
%   N11:0  PROC_STATE  "STATE The current state of the process" %
%   N9:11  PROC_PURIFY_A  "STATE Process Purify A" %
%   I:4.4  ADS_A_BED_TEMP  "TC6" %
%   N12:24  LT_INLET_GAS_WRN_SP %
%   N9:12  PROC_PURIFY_B  "STATE Process Purify B" %
%   I:4.6  ADS_B_BED_TEMP  "TC8" %
%   N7:3/4  LT_IN_GAS_WRN_EN %
%   T4:73  LT_IN_GAS_WRN_TMR %
%   N12:17/1  LT_INLET_GAS_WARN %

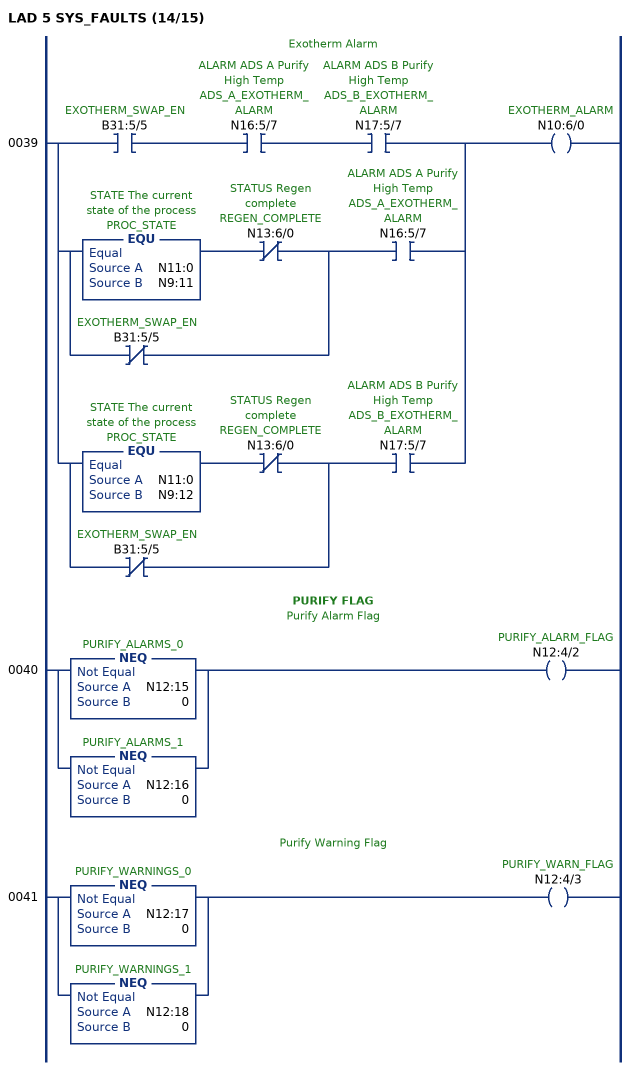
% Rung: 39 %
% Exotherm Alarm %
SOR BST XIC B31:5/5 XIC N16:5/7 XIC N17:5/7 NXB BST EQU N11:0 N9:11 XIO N13:6/0 NXB XIO B31:5/5 BND XIC N16:5/7 NXB BST EQU N11:0 N9:12 XIO N13:6/0 NXB XIO B31:5/5 BND XIC N17:5/7 BND OTE N10:6/0 EOR
%   B31:5/5  EXOTHERM_SWAP_EN %
%   N16:5/7  ADS_A_EXOTHERM_ALARM  "ALARM ADS A Purify High Temp" %
%   N17:5/7  ADS_B_EXOTHERM_ALARM  "ALARM ADS B Purify High Temp" %
%   N11:0  PROC_STATE  "STATE The current state of the process" %
%   N9:11  PROC_PURIFY_A  "STATE Process Purify A" %
%   N13:6/0  REGEN_COMPLETE  "STATUS Regen complete" %
%   N9:12  PROC_PURIFY_B  "STATE Process Purify B" %
%   N10:6/0  EXOTHERM_ALARM %
% Rung: 40 %
% TITLE: PURIFY FLAG %
% Purify Alarm Flag %
SOR BST NEQ N12:15 0 NXB NEQ N12:16 0 BND OTE N12:4/2 EOR
%   N12:15  PURIFY_ALARMS_0 %
%   N12:16  PURIFY_ALARMS_1 %
%   N12:4/2  PURIFY_ALARM_FLAG %
% Rung: 41 %
% Purify Warning Flag %
SOR BST NEQ N12:17 0 NXB NEQ N12:18 0 BND OTE N12:4/3 EOR
%   N12:17  PURIFY_WARNINGS_0 %
%   N12:18  PURIFY_WARNINGS_1 %
%   N12:4/3  PURIFY_WARN_FLAG %

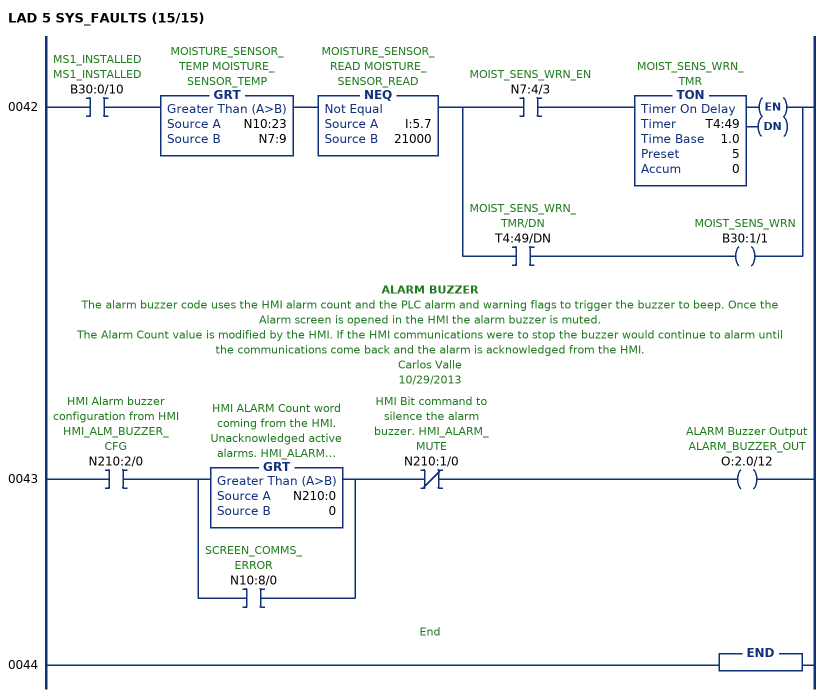
% Rung: 42 %
SOR XIC B30:0/10 GRT N10:23 N7:9 NEQ I:5.7 21000 BST XIC N7:4/3 TON T4:49 1.0 5 0 NXB XIC T4:49/DN OTE B30:1/1 BND EOR
%   B30:0/10  MS1_INSTALLED  "MS1_INSTALLED" %
%   N10:23  MOISTURE_SENSOR_TEMP  "MOISTURE_SENSOR_TEMP" %
%   N7:9  MOIST_SENS_WRN_SETP %
%   I:5.7  MOISTURE_SENSOR_READ  "MOISTURE_SENSOR_READ" %
%   N7:4/3  MOIST_SENS_WRN_EN %
%   T4:49  MOIST_SENS_WRN_TMR %
%   B30:1/1  MOIST_SENS_WRN %
% Rung: 43 %
% TITLE: ALARM BUZZER %
% The alarm buzzer code uses the HMI alarm count and the PLC alarm and warning flags to trigger the buzzer to beep. Once the Alarm screen is opened in the HMI the alarm buzzer is muted.
% The Alarm Count value is modified by the HMI. If the HMI communications were to stop the buzzer would continue to alarm until the communications come back and the alarm is acknowledged from the HMI.
% Carlos Valle
% 10/29/2013 %
SOR XIC N210:2/0 BST GRT N210:0 0 NXB XIC N10:8/0 BND XIO N210:1/0 OTE O:2.0/12 EOR
%   N210:2/0  HMI_ALM_BUZZER_CFG  "HMI Alarm buzzer configuration from HMI" %
%   N210:0  HMI_ALARM_COUNT  "HMI ALARM Count word coming from the HMI. Unacknowledged active alarms." %
%   N10:8/0  SCREEN_COMMS_ERROR %
%   N210:1/0  HMI_ALARM_MUTE  "HMI Bit command to silence the alarm buzzer." %
%   O:2.0/12  ALARM_BUZZER_OUT  "ALARM Buzzer Output" %
% Rung: 44 %
% End %
SOR END EOR

LADDER 6 "SYSTEM"    % Controls the system %
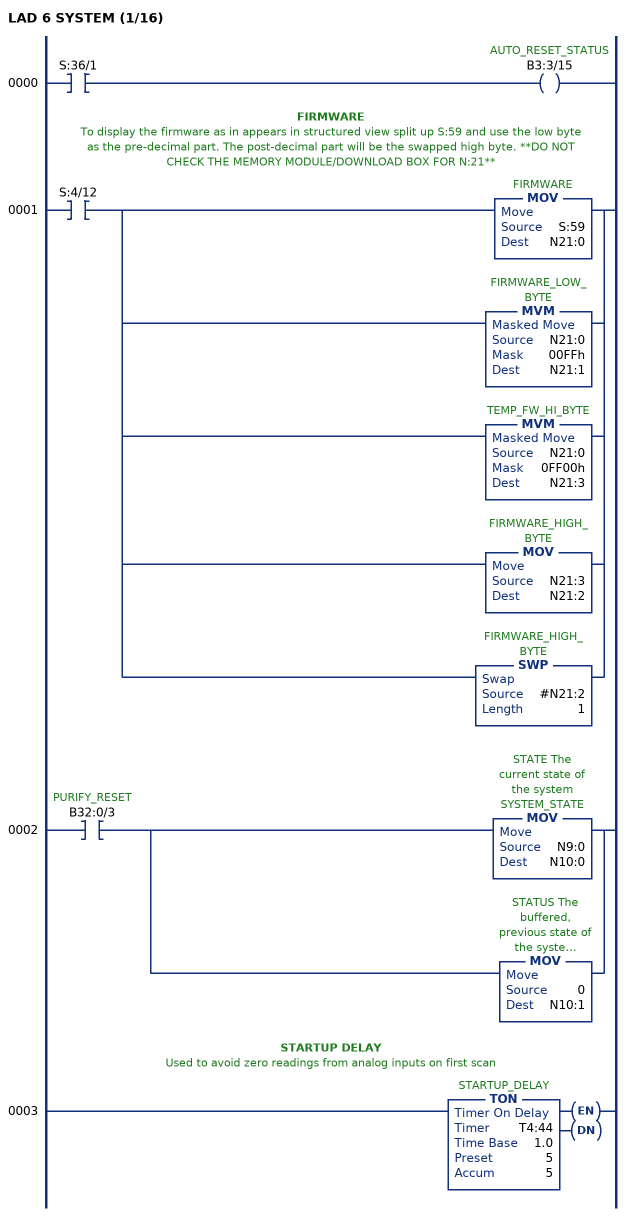
% Rung: 0 %
SOR XIC S:36/1 OTE B3:3/15 EOR
%   B3:3/15  AUTO_RESET_STATUS %
% Rung: 1 %
% TITLE: FIRMWARE %
% To display the firmware as in appears in structured view split up S:59 and use the low byte as the pre-decimal part. The post-decimal part will be the swapped high byte. **DO NOT CHECK THE MEMORY MODULE/DOWNLOAD BOX FOR N:21** %
SOR XIC S:4/12 BST MOV S:59 N21:0 NXB MVM N21:0 00FFh N21:1 NXB MVM N21:0 0FF00h N21:3 NXB MOV N21:3 N21:2 NXB SWP #N21:2 1 BND EOR
%   S:59  "Operating System FRN" %
%   N21:0  FIRMWARE %
%   N21:1  FIRMWARE_LOW_BYTE %
%   N21:3  TEMP_FW_HI_BYTE %
%   N21:2  FIRMWARE_HIGH_BYTE %
% Rung: 2 %
SOR XIC B32:0/3 BST MOV N9:0 N10:0 NXB MOV 0 N10:1 BND EOR
%   B32:0/3  PURIFY_RESET %
%   N9:0  SYSTEM_STANDBY  "STATE System Standby" %
%   N10:0  SYSTEM_STATE  "STATE The current state of the system" %
%   N10:1  SYSTEM_BUFFER  "STATUS The buffered, previous state of the system" %
% Rung: 3 %
% TITLE: STARTUP DELAY %
% Used to avoid zero readings from analog inputs on first scan %
SOR TON T4:44 1.0 5 5 EOR
%   T4:44  STARTUP_DELAY %

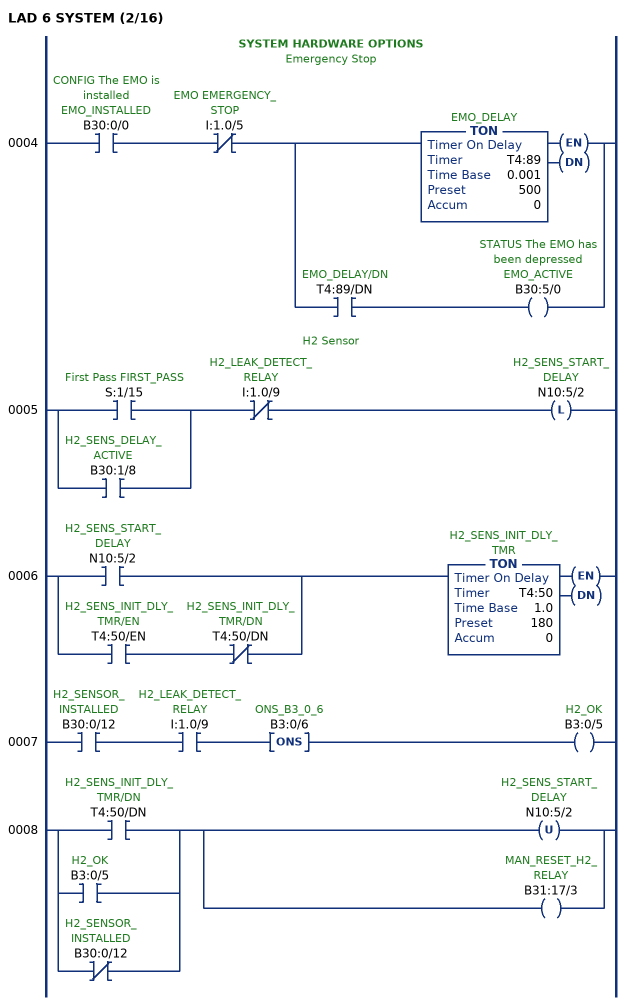
% Rung: 4 %
% TITLE: SYSTEM HARDWARE OPTIONS %
% Emergency Stop %
SOR XIC B30:0/0 XIO I:1.0/5 BST TON T4:89 0.001 500 0 NXB XIC T4:89/DN OTE B30:5/0 BND EOR
%   B30:0/0  EMO_INSTALLED  "CONFIG The EMO is installed" %
%   I:1.0/5  EMERGENCY_STOP  "EMO" %
%   T4:89  EMO_DELAY %
%   B30:5/0  EMO_ACTIVE  "STATUS The EMO has been depressed" %
% Rung: 5 %
% H2 Sensor %
SOR BST XIC S:1/15 NXB XIC B30:1/8 BND XIO I:1.0/9 OTL N10:5/2 EOR
%   S:1/15  FIRST_PASS  "First Pass" %
%   B30:1/8  H2_SENS_DELAY_ACTIVE %
%   I:1.0/9  H2_LEAK_DETECT_RELAY %
%   N10:5/2  H2_SENS_START_DELAY %
% Rung: 6 %
SOR BST XIC N10:5/2 NXB XIC T4:50/EN XIO T4:50/DN BND TON T4:50 1.0 180 0 EOR
%   N10:5/2  H2_SENS_START_DELAY %
%   T4:50  H2_SENS_INIT_DLY_TMR %
% Rung: 7 %
SOR XIC B30:0/12 XIC I:1.0/9 ONS B3:0/6 OTE B3:0/5 EOR
%   B30:0/12  H2_SENSOR_INSTALLED %
%   I:1.0/9  H2_LEAK_DETECT_RELAY %
%   B3:0/6  ONS_B3_0_6 %
%   B3:0/5  H2_OK %
% Rung: 8 %
SOR BST XIC T4:50/DN NXB XIC B3:0/5 NXB XIO B30:0/12 BND BST OTU N10:5/2 NXB OTE B31:17/3 BND EOR
%   T4:50  H2_SENS_INIT_DLY_TMR %
%   B3:0/5  H2_OK %
%   B30:0/12  H2_SENSOR_INSTALLED %
%   N10:5/2  H2_SENS_START_DELAY %
%   B31:17/3  MAN_RESET_H2_RELAY %

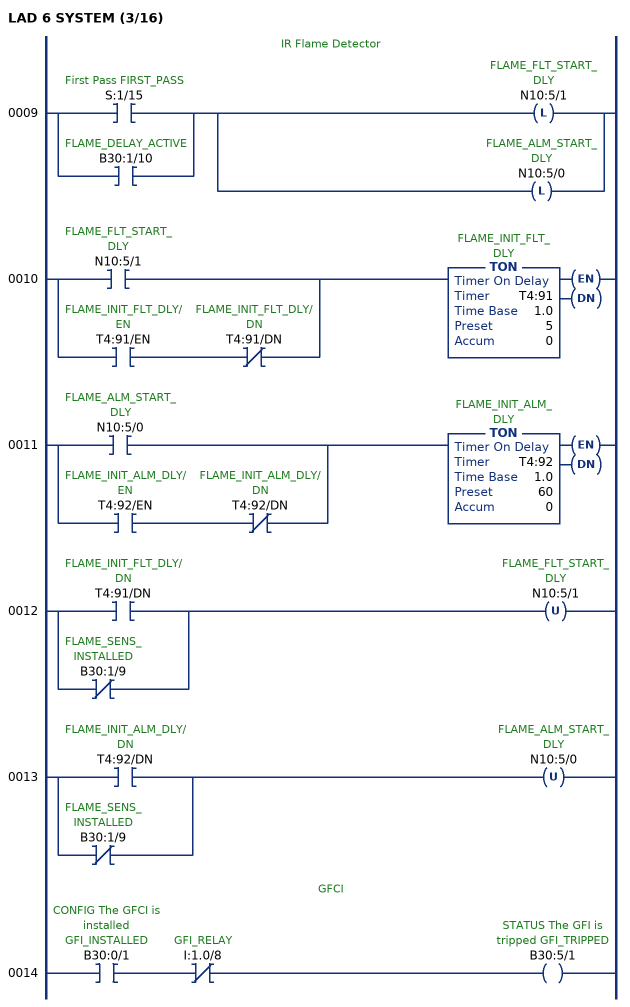
% Rung: 9 %
% IR Flame Detector %
SOR BST XIC S:1/15 NXB XIC B30:1/10 BND BST OTL N10:5/1 NXB OTL N10:5/0 BND EOR
%   S:1/15  FIRST_PASS  "First Pass" %
%   B30:1/10  FLAME_DELAY_ACTIVE %
%   N10:5/1  FLAME_FLT_START_DLY %
%   N10:5/0  FLAME_ALM_START_DLY %
% Rung: 10 %
SOR BST XIC N10:5/1 NXB XIC T4:91/EN XIO T4:91/DN BND TON T4:91 1.0 5 0 EOR
%   N10:5/1  FLAME_FLT_START_DLY %
%   T4:91  FLAME_INIT_FLT_DLY %
% Rung: 11 %
SOR BST XIC N10:5/0 NXB XIC T4:92/EN XIO T4:92/DN BND TON T4:92 1.0 60 0 EOR
%   N10:5/0  FLAME_ALM_START_DLY %
%   T4:92  FLAME_INIT_ALM_DLY %
% Rung: 12 %
SOR BST XIC T4:91/DN NXB XIO B30:1/9 BND OTU N10:5/1 EOR
%   T4:91  FLAME_INIT_FLT_DLY %
%   B30:1/9  FLAME_SENS_INSTALLED %
%   N10:5/1  FLAME_FLT_START_DLY %
% Rung: 13 %
SOR BST XIC T4:92/DN NXB XIO B30:1/9 BND OTU N10:5/0 EOR
%   T4:92  FLAME_INIT_ALM_DLY %
%   B30:1/9  FLAME_SENS_INSTALLED %
%   N10:5/0  FLAME_ALM_START_DLY %
% Rung: 14 %
% GFCI %
SOR XIC B30:0/1 XIO I:1.0/8 OTE B30:5/1 EOR
%   B30:0/1  GFI_INSTALLED  "CONFIG The GFCI is installed" %
%   I:1.0/8  GFI_RELAY %
%   B30:5/1  GFI_TRIPPED  "STATUS The GFI is tripped" %

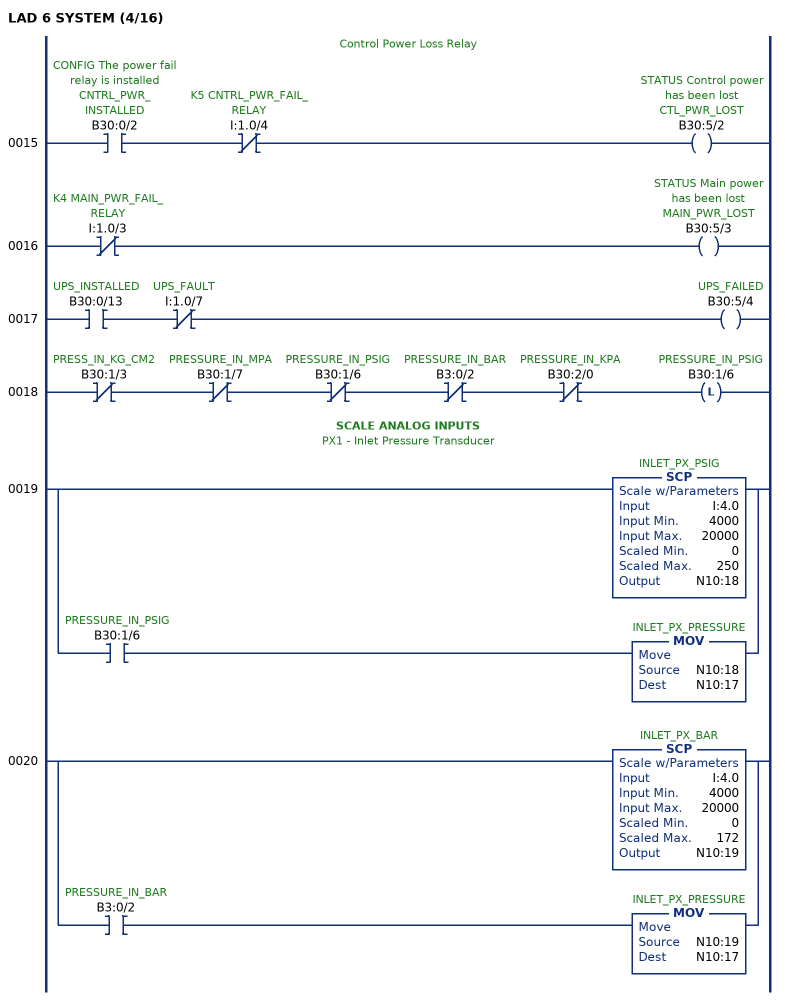
% Rung: 15 %
% Control Power Loss Relay %
SOR XIC B30:0/2 XIO I:1.0/4 OTE B30:5/2 EOR
%   B30:0/2  CNTRL_PWR_INSTALLED  "CONFIG The power fail relay is installed" %
%   I:1.0/4  CNTRL_PWR_FAIL_RELAY  "K5" %
%   B30:5/2  CTL_PWR_LOST  "STATUS Control power has been lost" %
% Rung: 16 %
SOR XIO I:1.0/3 OTE B30:5/3 EOR
%   I:1.0/3  MAIN_PWR_FAIL_RELAY  "K4" %
%   B30:5/3  MAIN_PWR_LOST  "STATUS Main power has been lost" %
% Rung: 17 %
SOR XIC B30:0/13 XIO I:1.0/7 OTE B30:5/4 EOR
%   B30:0/13  UPS_INSTALLED %
%   I:1.0/7  UPS_FAULT %
%   B30:5/4  UPS_FAILED %
% Rung: 18 %
SOR XIO B30:1/3 XIO B30:1/7 XIO B30:1/6 XIO B3:0/2 XIO B30:2/0 OTL B30:1/6 EOR
%   B30:1/3  PRESS_IN_KG_CM2 %
%   B30:1/7  PRESSURE_IN_MPA %
%   B30:1/6  PRESSURE_IN_PSIG %
%   B3:0/2  PRESSURE_IN_BAR %
%   B30:2/0  PRESSURE_IN_KPA %
% Rung: 19 %
% TITLE: SCALE ANALOG INPUTS %
% PX1 - Inlet Pressure Transducer %
SOR BST SCP I:4.0 4000 20000 0 250 N10:18 NXB XIC B30:1/6 MOV N10:18 N10:17 BND EOR
%   I:4.0  INLET_PX_READING  "PX-1" %
%   N10:18  INLET_PX_PSIG %
%   B30:1/6  PRESSURE_IN_PSIG %
%   N10:17  INLET_PX_PRESSURE %
% Rung: 20 %
SOR BST SCP I:4.0 4000 20000 0 172 N10:19 NXB XIC B3:0/2 MOV N10:19 N10:17 BND EOR
%   I:4.0  INLET_PX_READING  "PX-1" %
%   N10:19  INLET_PX_BAR %
%   B3:0/2  PRESSURE_IN_BAR %
%   N10:17  INLET_PX_PRESSURE %

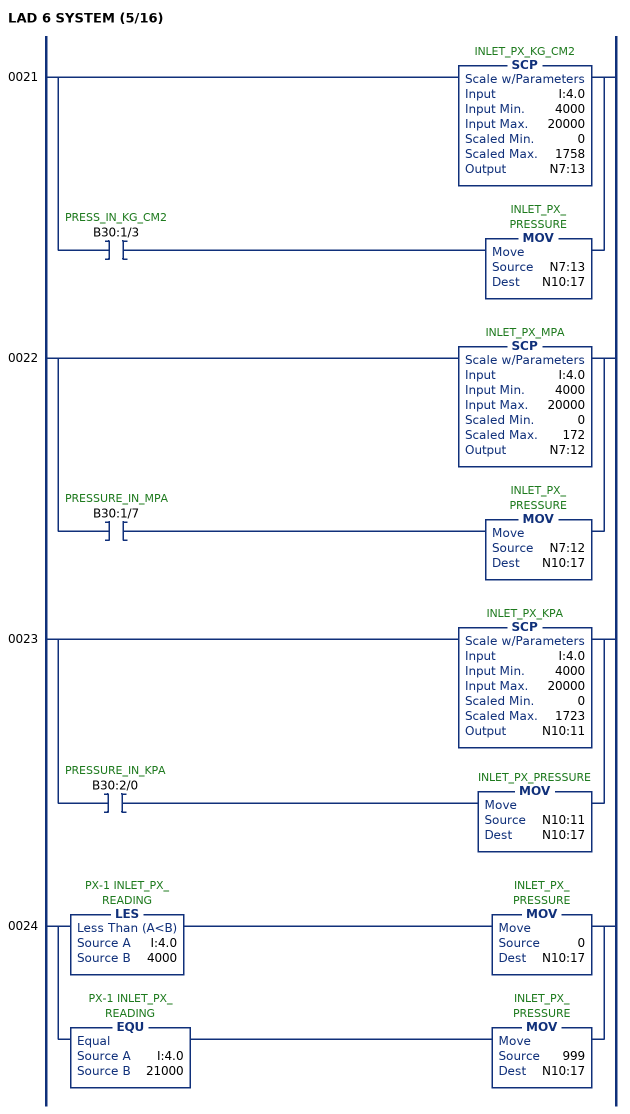
% Rung: 21 %
SOR BST SCP I:4.0 4000 20000 0 1758 N7:13 NXB XIC B30:1/3 MOV N7:13 N10:17 BND EOR
%   I:4.0  INLET_PX_READING  "PX-1" %
%   N7:13  INLET_PX_KG_CM2 %
%   B30:1/3  PRESS_IN_KG_CM2 %
%   N10:17  INLET_PX_PRESSURE %
% Rung: 22 %
SOR BST SCP I:4.0 4000 20000 0 172 N7:12 NXB XIC B30:1/7 MOV N7:12 N10:17 BND EOR
%   I:4.0  INLET_PX_READING  "PX-1" %
%   N7:12  INLET_PX_MPA %
%   B30:1/7  PRESSURE_IN_MPA %
%   N10:17  INLET_PX_PRESSURE %
% Rung: 23 %
SOR BST SCP I:4.0 4000 20000 0 1723 N10:11 NXB XIC B30:2/0 MOV N10:11 N10:17 BND EOR
%   I:4.0  INLET_PX_READING  "PX-1" %
%   N10:11  INLET_PX_KPA %
%   B30:2/0  PRESSURE_IN_KPA %
%   N10:17  INLET_PX_PRESSURE %
% Rung: 24 %
SOR BST LES I:4.0 4000 MOV 0 N10:17 NXB EQU I:4.0 21000 MOV 999 N10:17 BND EOR
%   I:4.0  INLET_PX_READING  "PX-1" %
%   N10:17  INLET_PX_PRESSURE %

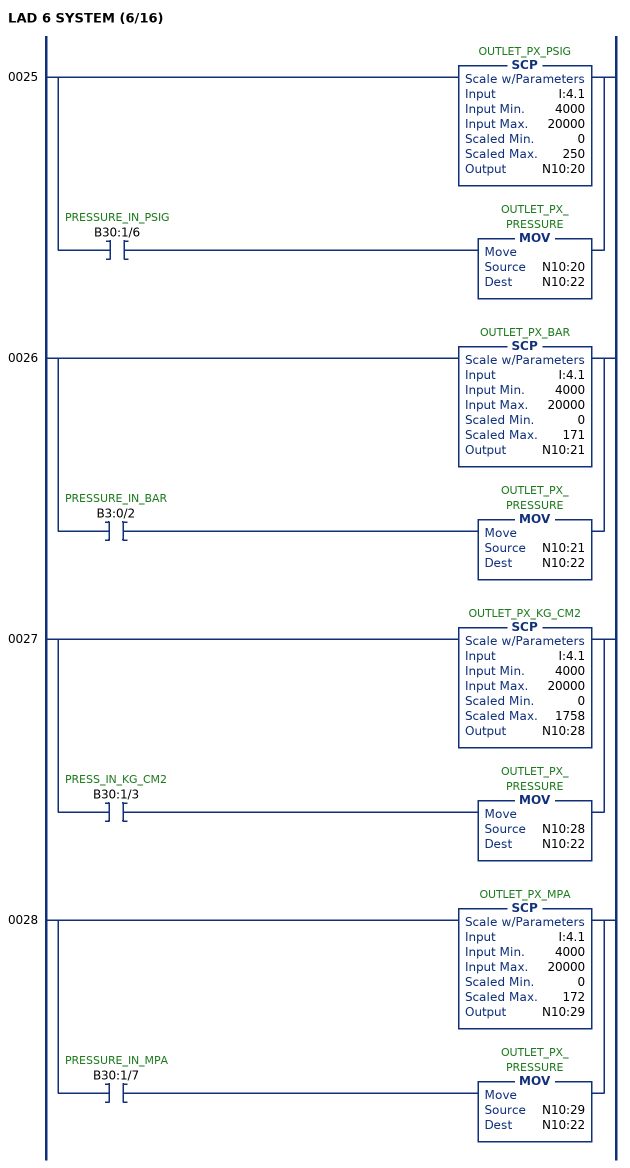
% Rung: 25 %
SOR BST SCP I:4.1 4000 20000 0 250 N10:20 NXB XIC B30:1/6 MOV N10:20 N10:22 BND EOR
%   I:4.1  OUTLET_PX_READING  "PX-2" %
%   N10:20  OUTLET_PX_PSIG %
%   B30:1/6  PRESSURE_IN_PSIG %
%   N10:22  OUTLET_PX_PRESSURE %
% Rung: 26 %
SOR BST SCP I:4.1 4000 20000 0 171 N10:21 NXB XIC B3:0/2 MOV N10:21 N10:22 BND EOR
%   I:4.1  OUTLET_PX_READING  "PX-2" %
%   N10:21  OUTLET_PX_BAR %
%   B3:0/2  PRESSURE_IN_BAR %
%   N10:22  OUTLET_PX_PRESSURE %
% Rung: 27 %
SOR BST SCP I:4.1 4000 20000 0 1758 N10:28 NXB XIC B30:1/3 MOV N10:28 N10:22 BND EOR
%   I:4.1  OUTLET_PX_READING  "PX-2" %
%   N10:28  OUTLET_PX_KG_CM2 %
%   B30:1/3  PRESS_IN_KG_CM2 %
%   N10:22  OUTLET_PX_PRESSURE %
% Rung: 28 %
SOR BST SCP I:4.1 4000 20000 0 172 N10:29 NXB XIC B30:1/7 MOV N10:29 N10:22 BND EOR
%   I:4.1  OUTLET_PX_READING  "PX-2" %
%   N10:29  OUTLET_PX_MPA %
%   B30:1/7  PRESSURE_IN_MPA %
%   N10:22  OUTLET_PX_PRESSURE %

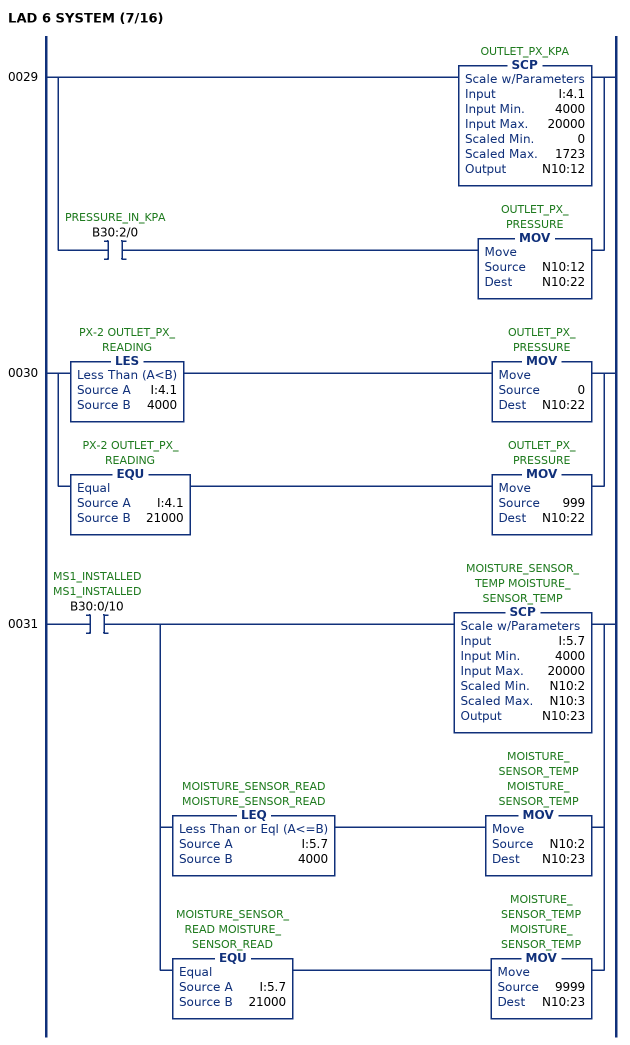
% Rung: 29 %
SOR BST SCP I:4.1 4000 20000 0 1723 N10:12 NXB XIC B30:2/0 MOV N10:12 N10:22 BND EOR
%   I:4.1  OUTLET_PX_READING  "PX-2" %
%   N10:12  OUTLET_PX_KPA %
%   B30:2/0  PRESSURE_IN_KPA %
%   N10:22  OUTLET_PX_PRESSURE %
% Rung: 30 %
SOR BST LES I:4.1 4000 MOV 0 N10:22 NXB EQU I:4.1 21000 MOV 999 N10:22 BND EOR
%   I:4.1  OUTLET_PX_READING  "PX-2" %
%   N10:22  OUTLET_PX_PRESSURE %
% Rung: 31 %
SOR XIC B30:0/10 BST SCP I:5.7 4000 20000 N10:2 N10:3 N10:23 NXB LEQ I:5.7 4000 MOV N10:2 N10:23 NXB EQU I:5.7 21000 MOV 9999 N10:23 BND EOR
%   B30:0/10  MS1_INSTALLED  "MS1_INSTALLED" %
%   I:5.7  MOISTURE_SENSOR_READ  "MOISTURE_SENSOR_READ" %
%   N10:2  MOISTURE_SENSOR_MIN %
%   N10:3  MOISTURE_SENSOR_MAX %
%   N10:23  MOISTURE_SENSOR_TEMP  "MOISTURE_SENSOR_TEMP" %

